// TIA Portal V17 export
// export: Created 2025-11-18T11:18:45.6774883Z, ExportSetting WithDefaults, DisplayName Totally Integrated Automation Portal, DisplayVersion V17 Update 8, DisplayName TIA Portal Openness, DisplayVersion V17 Update 8, DisplayName TIA Portal Version Control Interface, DisplayVersion V17, DisplayName STEP 7 Professional, DisplayVersion V17 Update 8, DisplayName STEP 7 Safety, DisplayVersion V17 Update 6, DisplayName WinCC Advanced, DisplayVersion V17 Update 8
FUNCTION_BLOCK "PLC_VLC_Connection_TCP-IP"   // FB1, LAD
{ S7_Optimized_Access := 'TRUE' }
VERSION : 0.1
// stored: AutoNumber true, IsIECCheckEnabled false, IsRetainMemResEnabled false, MemoryReserve 100, SetENOAutomatically false, UDAEnableTagReadback false
   VAR_INPUT
      xFirstScan : Bool;
      xAlwaysTRUE : Bool;
      xDataReceiveOn : Bool;
   END_VAR
   VAR_OUTPUT
      Connection_OK : Bool;
      Connected : Bool;
      Started : Bool;
      Paused : Bool;
      EndOfFile : Bool;
   END_VAR
   VAR_IN_OUT
      xSendRequest : Bool;
      xCommandStart : Bool;
      xCommandStop : Bool;
      xCommandReset : Bool;
      xCommandPause : Bool;
      xCommandResume : Bool;
      xCommandRewind0 : Bool;
      xCommandRewindX : Bool;
      xReconnect : Bool;
   END_VAR
   VAR
      TCON_Instance { S7_SetPoint := 'True'} : TCON;
      TCON : Struct
         REC : Bool;
         DONE : Bool;
         BUSY : Bool;
         ERROR : Bool;
         DONE_Memo : Bool;
         STATUS : Word;
      END_STRUCT;
      TDISCON : Struct
         REQ : Bool;
         DONE : Bool;
         BUSY : Bool;
         ERROR : Bool;
         STATUS : Word;
      END_STRUCT;
      TSEND : Struct
         REQ : Bool;
         DONE : Bool;
         BUSY : Bool;
         ERROR : Bool;
         DONE_Memo : Bool;
         STATUS : Word;
      END_STRUCT;
      TRCV : Struct
         EN_R : Bool;
         NDR : Bool;
         BUSY : Bool;
         ERROR : Bool;
         STATUS : Word;
         RCVD_LENGTH : UDInt;
      END_STRUCT;
      TDISCON_DB { S7_SetPoint := 'True'} : TDISCON;
      TSEND_Instance { S7_SetPoint := 'True'} : TSEND;
      TRCV_Instance { S7_SetPoint := 'True'} : TRCV;
      Variables : Struct
         ConnectRequest : Bool;
         DisconnectRequest : Bool;
         Reconect : Bool;
         SendString : String;
         DataToSend : String;
         Heartbeat0 : Bool;
         Heartbeat1 : Bool;
         Heartbeat_ConnectionOK : Bool;
         Receive : Array[0..20] of Char;
         ReceivedString : String;
      END_STRUCT;
      Pulses { S7_SetPoint := 'True'} : Array[0..10] of Bool;
      IEC_Timer_SendData { S7_SetPoint := 'True'} : TP_TIME;
      IEC_Timer_SendRequestToLong { S7_SetPoint := 'True'} : TON_TIME;
      IEC_TimerReconnect { S7_SetPoint := 'True'} : TON_TIME;
      IEC_Timer_ReadDelayAfterConnect { S7_SetPoint := 'True'} : TON_TIME;
      TON_HB_1 { S7_SetPoint := 'True'} : TON_TIME;
      TON_HB_2 { S7_SetPoint := 'True'} : TON_TIME;
      TON_HB_3 { S7_SetPoint := 'True'} : TON_TIME;
      ReconnectTimer { S7_SetPoint := 'True'} : TON_TIME;
      RecoonectTimer2 { S7_SetPoint := 'True'} : TON_TIME;
      pulse : Bool;
      pulse2 : Bool;
      resetTimera : Bool;
      pulse3 : Bool;
   END_VAR
   VAR_TEMP
      tempInt : Int;
   END_VAR
   VAR CONSTANT
      EndPoint : String := '\n';
   END_VAR
   VAR_TEMP   // added for the SCL form of the ladder/FBD networks
      _w1 : Bool;
      _w2 : Bool;
      _w3 : Bool;
      _w4 : Bool;
      _w5 : Bool;
      _w6 : Bool;
      _w7 : Bool;
      _w8 : Bool;
      _w9 : Bool;
      _w10 : Bool;
      _w11 : Bool;
      _w12 : Bool;
      _w13 : Bool;
      _w14 : Bool;
      _w15 : Bool;
      _w16 : Bool;
   END_VAR
BEGIN

REGION Network 1: Connection Init
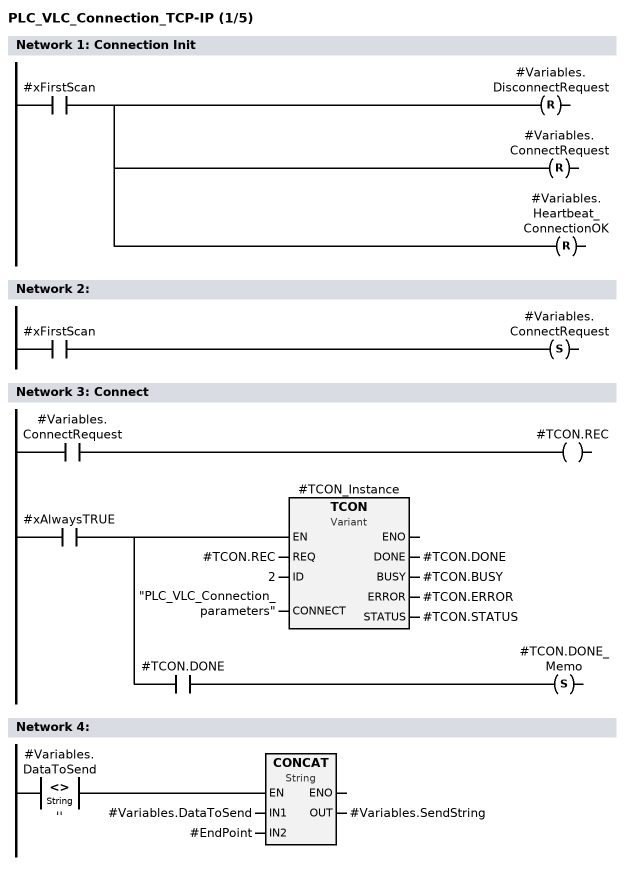
   RUNG wire#powerrail
      Contact( #xFirstScan )
      wire#w1
      R_Coil( #Variables.DisconnectRequest )
   END_RUNG
   RUNG wire#w1
      R_Coil( #Variables.ConnectRequest )
   END_RUNG
   RUNG wire#w1
      R_Coil( #Variables.Heartbeat_ConnectionOK )
   END_RUNG
   // the same network as SCL:
   IF #xFirstScan THEN
       #Variables.DisconnectRequest := FALSE;
       #Variables.ConnectRequest := FALSE;
       #Variables.Heartbeat_ConnectionOK := FALSE;
   END_IF;
END_REGION

REGION Network 2
   RUNG wire#powerrail
      Contact( #xFirstScan )
      S_Coil( #Variables.ConnectRequest )
   END_RUNG
   // the same network as SCL:
   IF #xFirstScan THEN #Variables.ConnectRequest := TRUE; END_IF;
END_REGION

REGION Network 3: Connect
   RUNG wire#powerrail
      Contact( #Variables.ConnectRequest )
      Coil( #TCON.REC )
   END_RUNG
   RUNG wire#powerrail
      Contact( #xAlwaysTRUE )
      wire#w1
      { S7_Templates := "[con_type := Variant, id_type := CONN_OUC]" } #TCON_Instance.TCON(REQ := #TCON.REC, ID := 2, CONNECT := "PLC_VLC_Connection_parameters", DONE => #TCON.DONE, BUSY => #TCON.BUSY, ERROR => #TCON.ERROR, STATUS => #TCON.STATUS)
   END_RUNG
   RUNG wire#w1
      Contact( #TCON.DONE )
      S_Coil( #TCON.DONE_Memo )
   END_RUNG
   // the same network as SCL:
   #TCON.REC := #Variables.ConnectRequest;
   IF #xAlwaysTRUE THEN
       #TCON_Instance(REQ := #TCON.REC,   // TCON
                      ID := 2,
                      CONNECT := "PLC_VLC_Connection_parameters",
                      DONE => #TCON.DONE,
                      BUSY => #TCON.BUSY,
                      ERROR => #TCON.ERROR,
                      STATUS => #TCON.STATUS);
   END_IF;
   IF #xAlwaysTRUE AND #TCON.DONE THEN #TCON.DONE_Memo := TRUE; END_IF;
END_REGION

REGION Network 4
   RUNG wire#powerrail
      { S7_Templates := "SrcType := String" } NE_Contact(in1 := #Variables.DataToSend, in2 := '')
      { S7_Templates := "[card := 2, str_type := String]" } CONCAT(IN1 := #Variables.DataToSend, IN2 := #EndPoint, OUT => #Variables.SendString)
   END_RUNG
   // the same network as SCL:
   IF #Variables.DataToSend <> '' THEN
       CONCAT(IN1 := #Variables.DataToSend, IN2 := #EndPoint, OUT => #Variables.SendString);
   END_IF;
END_REGION

REGION Network 5
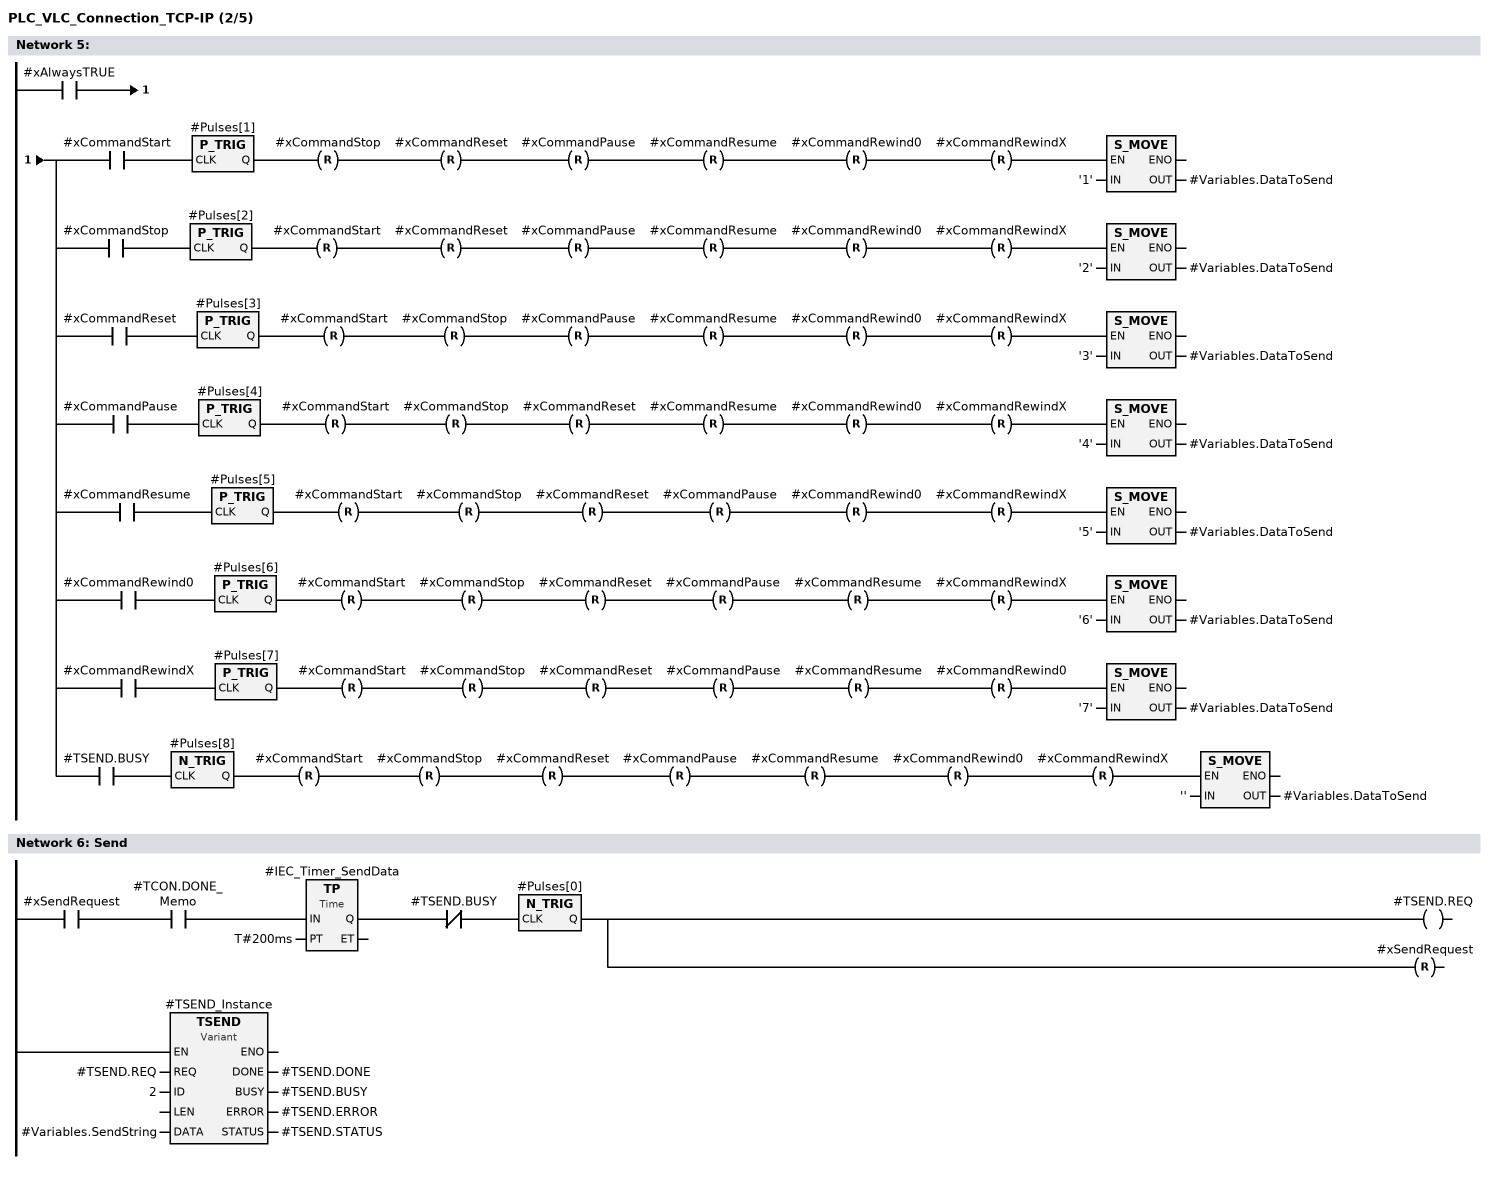
   RUNG wire#powerrail
      Contact( #xAlwaysTRUE )
      wire#w1
      Contact( #xCommandStart )
      P_Trig( #Pulses[1] )
      R_Coil( #xCommandStop )
      R_Coil( #xCommandReset )
      R_Coil( #xCommandPause )
      R_Coil( #xCommandResume )
      R_Coil( #xCommandRewind0 )
      R_Coil( #xCommandRewindX )
      S_Move(in := '1', out => #Variables.DataToSend)
   END_RUNG
   RUNG wire#w1
      Contact( #xCommandStop )
      P_Trig( #Pulses[2] )
      R_Coil( #xCommandStart )
      R_Coil( #xCommandReset )
      R_Coil( #xCommandPause )
      R_Coil( #xCommandResume )
      R_Coil( #xCommandRewind0 )
      R_Coil( #xCommandRewindX )
      S_Move(in := '2', out => #Variables.DataToSend)
   END_RUNG
   RUNG wire#w1
      Contact( #xCommandReset )
      P_Trig( #Pulses[3] )
      R_Coil( #xCommandStart )
      R_Coil( #xCommandStop )
      R_Coil( #xCommandPause )
      R_Coil( #xCommandResume )
      R_Coil( #xCommandRewind0 )
      R_Coil( #xCommandRewindX )
      S_Move(in := '3', out => #Variables.DataToSend)
   END_RUNG
   RUNG wire#w1
      Contact( #xCommandPause )
      P_Trig( #Pulses[4] )
      R_Coil( #xCommandStart )
      R_Coil( #xCommandStop )
      R_Coil( #xCommandReset )
      R_Coil( #xCommandResume )
      R_Coil( #xCommandRewind0 )
      R_Coil( #xCommandRewindX )
      S_Move(in := '4', out => #Variables.DataToSend)
   END_RUNG
   RUNG wire#w1
      Contact( #xCommandResume )
      P_Trig( #Pulses[5] )
      R_Coil( #xCommandStart )
      R_Coil( #xCommandStop )
      R_Coil( #xCommandReset )
      R_Coil( #xCommandPause )
      R_Coil( #xCommandRewind0 )
      R_Coil( #xCommandRewindX )
      S_Move(in := '5', out => #Variables.DataToSend)
   END_RUNG
   RUNG wire#w1
      Contact( #xCommandRewind0 )
      P_Trig( #Pulses[6] )
      R_Coil( #xCommandStart )
      R_Coil( #xCommandStop )
      R_Coil( #xCommandReset )
      R_Coil( #xCommandPause )
      R_Coil( #xCommandResume )
      R_Coil( #xCommandRewindX )
      S_Move(in := '6', out => #Variables.DataToSend)
   END_RUNG
   RUNG wire#w1
      Contact( #xCommandRewindX )
      P_Trig( #Pulses[7] )
      R_Coil( #xCommandStart )
      R_Coil( #xCommandStop )
      R_Coil( #xCommandReset )
      R_Coil( #xCommandPause )
      R_Coil( #xCommandResume )
      R_Coil( #xCommandRewind0 )
      S_Move(in := '7', out => #Variables.DataToSend)
   END_RUNG
   RUNG wire#w1
      Contact( #TSEND.BUSY )
      N_Trig( #Pulses[8] )
      R_Coil( #xCommandStart )
      R_Coil( #xCommandStop )
      R_Coil( #xCommandReset )
      R_Coil( #xCommandPause )
      R_Coil( #xCommandResume )
      R_Coil( #xCommandRewind0 )
      R_Coil( #xCommandRewindX )
      S_Move(in := '', out => #Variables.DataToSend)
   END_RUNG
   // the same network as SCL:
   #_w1 := #xAlwaysTRUE AND #xCommandStart;
   #_w2 := #_w1 AND NOT #Pulses[1];   // rising edge
   #Pulses[1] := #_w1;
   IF #_w2 THEN
       #xCommandStop := FALSE;
       #xCommandReset := FALSE;
       #xCommandPause := FALSE;
       #xCommandResume := FALSE;
       #xCommandRewind0 := FALSE;
       #xCommandRewindX := FALSE;
       #Variables.DataToSend := '1';
   END_IF;
   #_w3 := #xAlwaysTRUE AND #xCommandStop;
   #_w4 := #_w3 AND NOT #Pulses[2];   // rising edge
   #Pulses[2] := #_w3;
   IF #_w4 THEN
       #xCommandStart := FALSE;
       #xCommandReset := FALSE;
       #xCommandPause := FALSE;
       #xCommandResume := FALSE;
       #xCommandRewind0 := FALSE;
       #xCommandRewindX := FALSE;
       #Variables.DataToSend := '2';
   END_IF;
   #_w5 := #xAlwaysTRUE AND #xCommandReset;
   #_w6 := #_w5 AND NOT #Pulses[3];   // rising edge
   #Pulses[3] := #_w5;
   IF #_w6 THEN
       #xCommandStart := FALSE;
       #xCommandStop := FALSE;
       #xCommandPause := FALSE;
       #xCommandResume := FALSE;
       #xCommandRewind0 := FALSE;
       #xCommandRewindX := FALSE;
       #Variables.DataToSend := '3';
   END_IF;
   #_w7 := #xAlwaysTRUE AND #xCommandPause;
   #_w8 := #_w7 AND NOT #Pulses[4];   // rising edge
   #Pulses[4] := #_w7;
   IF #_w8 THEN
       #xCommandStart := FALSE;
       #xCommandStop := FALSE;
       #xCommandReset := FALSE;
       #xCommandResume := FALSE;
       #xCommandRewind0 := FALSE;
       #xCommandRewindX := FALSE;
       #Variables.DataToSend := '4';
   END_IF;
   #_w9 := #xAlwaysTRUE AND #xCommandResume;
   #_w10 := #_w9 AND NOT #Pulses[5];   // rising edge
   #Pulses[5] := #_w9;
   IF #_w10 THEN
       #xCommandStart := FALSE;
       #xCommandStop := FALSE;
       #xCommandReset := FALSE;
       #xCommandPause := FALSE;
       #xCommandRewind0 := FALSE;
       #xCommandRewindX := FALSE;
       #Variables.DataToSend := '5';
   END_IF;
   #_w11 := #xAlwaysTRUE AND #xCommandRewind0;
   #_w12 := #_w11 AND NOT #Pulses[6];   // rising edge
   #Pulses[6] := #_w11;
   IF #_w12 THEN
       #xCommandStart := FALSE;
       #xCommandStop := FALSE;
       #xCommandReset := FALSE;
       #xCommandPause := FALSE;
       #xCommandResume := FALSE;
       #xCommandRewindX := FALSE;
       #Variables.DataToSend := '6';
   END_IF;
   #_w13 := #xAlwaysTRUE AND #xCommandRewindX;
   #_w14 := #_w13 AND NOT #Pulses[7];   // rising edge
   #Pulses[7] := #_w13;
   IF #_w14 THEN
       #xCommandStart := FALSE;
       #xCommandStop := FALSE;
       #xCommandReset := FALSE;
       #xCommandPause := FALSE;
       #xCommandResume := FALSE;
       #xCommandRewind0 := FALSE;
       #Variables.DataToSend := '7';
   END_IF;
   #_w15 := #xAlwaysTRUE AND #TSEND.BUSY;
   #_w16 := NOT #_w15 AND #Pulses[8];   // falling edge
   #Pulses[8] := #_w15;
   IF #_w16 THEN
       #xCommandStart := FALSE;
       #xCommandStop := FALSE;
       #xCommandReset := FALSE;
       #xCommandPause := FALSE;
       #xCommandResume := FALSE;
       #xCommandRewind0 := FALSE;
       #xCommandRewindX := FALSE;
       #Variables.DataToSend := '';
   END_IF;
END_REGION

REGION Network 6: Send
   RUNG wire#powerrail
      Contact( #xSendRequest )
      Contact( #TCON.DONE_Memo )
      { S7_Templates := "time_type := Time" } #IEC_Timer_SendData.TP(pt := T#200ms, et =>)
      I_Contact( #TSEND.BUSY )
      N_Trig( #Pulses[0] )
      wire#w1
      Coil( #TSEND.REQ )
   END_RUNG
   RUNG wire#w1
      R_Coil( #xSendRequest )
   END_RUNG
   RUNG wire#powerrail
      { S7_Templates := "[data_type := Variant, len_type := UDInt, id_type := CONN_OUC]" } #TSEND_Instance.TSEND(REQ := #TSEND.REQ, ID := 2, LEN :=, DATA := #Variables.SendString, DONE => #TSEND.DONE, BUSY => #TSEND.BUSY, ERROR => #TSEND.ERROR, STATUS => #TSEND.STATUS)
   END_RUNG
   // the same network as SCL:
   #IEC_Timer_SendData(IN := #xSendRequest AND #TCON.DONE_Memo, PT := T#200ms);   // TP
   #_w1 := #IEC_Timer_SendData.Q AND NOT #TSEND.BUSY;
   #_w2 := NOT #_w1 AND #Pulses[0];   // falling edge
   #Pulses[0] := #_w1;
   #TSEND.REQ := #_w2;
   IF #_w2 THEN #xSendRequest := FALSE; END_IF;
   #TSEND_Instance(REQ := #TSEND.REQ,   // TSEND
                   ID := 2,
                   DATA := #Variables.SendString,
                   DONE => #TSEND.DONE,
                   BUSY => #TSEND.BUSY,
                   ERROR => #TSEND.ERROR,
                   STATUS => #TSEND.STATUS);
END_REGION

REGION Network 7: Receive
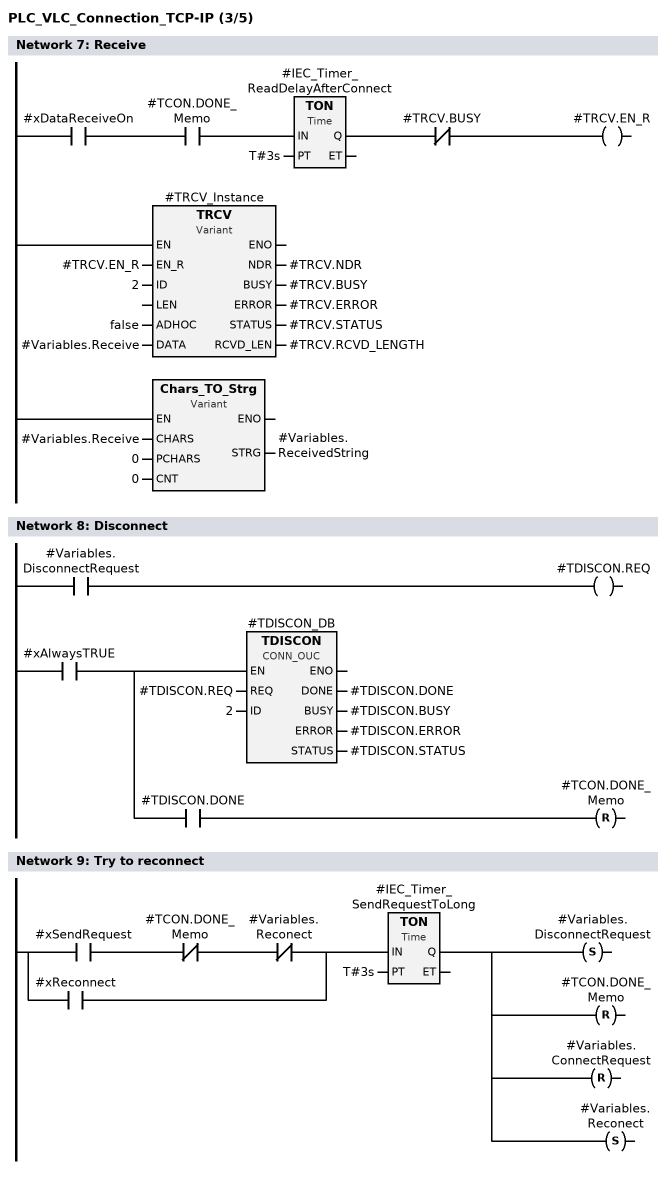
   RUNG wire#powerrail
      Contact( #xDataReceiveOn )
      Contact( #TCON.DONE_Memo )
      { S7_Templates := "time_type := Time" } #IEC_Timer_ReadDelayAfterConnect.TON(pt := T#3s, et =>)
      I_Contact( #TRCV.BUSY )
      Coil( #TRCV.EN_R )
   END_RUNG
   RUNG wire#powerrail
      { S7_Templates := "[card := 1, ptr_type := Variant, value_type := UDInt, id_type := CONN_OUC]" } #TRCV_Instance.TRCV(EN_R := #TRCV.EN_R, ID := 2, LEN :=, ADHOC := false, DATA := #Variables.Receive, NDR => #TRCV.NDR, BUSY => #TRCV.BUSY, ERROR => #TRCV.ERROR, STATUS => #TRCV.STATUS, RCVD_LEN => #TRCV.RCVD_LENGTH)
   END_RUNG
   RUNG wire#powerrail
      { S7_Templates := "[ptr_type := Variant, str_type := String]" } Chars_TO_Strg(Chars := #Variables.Receive, pChars := 0, Cnt := 0, Strg => #Variables.ReceivedString)
   END_RUNG
   // the same network as SCL:
   #IEC_Timer_ReadDelayAfterConnect(IN := #xDataReceiveOn AND #TCON.DONE_Memo, PT := T#3s);   // TON
   #TRCV.EN_R := #IEC_Timer_ReadDelayAfterConnect.Q AND NOT #TRCV.BUSY;
   #TRCV_Instance(EN_R := #TRCV.EN_R,   // TRCV
                  ID := 2,
                  ADHOC := false,
                  DATA := #Variables.Receive,
                  NDR => #TRCV.NDR,
                  BUSY => #TRCV.BUSY,
                  ERROR => #TRCV.ERROR,
                  STATUS => #TRCV.STATUS,
                  RCVD_LEN => #TRCV.RCVD_LENGTH);
   Chars_TO_Strg(Chars := #Variables.Receive, pChars := 0, Cnt := 0, Strg => #Variables.ReceivedString);
END_REGION

REGION Network 8: Disconnect
   RUNG wire#powerrail
      Contact( #Variables.DisconnectRequest )
      Coil( #TDISCON.REQ )
   END_RUNG
   RUNG wire#powerrail
      Contact( #xAlwaysTRUE )
      wire#w1
      { S7_Templates := "id_type := CONN_OUC" } #TDISCON_DB.TDISCON(REQ := #TDISCON.REQ, ID := 2, DONE => #TDISCON.DONE, BUSY => #TDISCON.BUSY, ERROR => #TDISCON.ERROR, STATUS => #TDISCON.STATUS)
   END_RUNG
   RUNG wire#w1
      Contact( #TDISCON.DONE )
      R_Coil( #TCON.DONE_Memo )
   END_RUNG
   // the same network as SCL:
   #TDISCON.REQ := #Variables.DisconnectRequest;
   IF #xAlwaysTRUE THEN
       #TDISCON_DB(REQ := #TDISCON.REQ,   // TDISCON
                   ID := 2,
                   DONE => #TDISCON.DONE,
                   BUSY => #TDISCON.BUSY,
                   ERROR => #TDISCON.ERROR,
                   STATUS => #TDISCON.STATUS);
   END_IF;
   IF #xAlwaysTRUE AND #TDISCON.DONE THEN #TCON.DONE_Memo := FALSE; END_IF;
END_REGION

REGION Network 9: Try to reconnect
   RUNG wire#powerrail
      Contact( #xSendRequest )
      I_Contact( #TCON.DONE_Memo )
      I_Contact( #Variables.Reconect )
      wire#w1
      { S7_Templates := "time_type := Time" } #IEC_Timer_SendRequestToLong.TON(pt := T#3s, et =>)
      wire#w2
      S_Coil( #Variables.DisconnectRequest )
   END_RUNG
   RUNG wire#powerrail
      Contact( #xReconnect )
   END_RUNG wire#w1
   RUNG wire#w2
      R_Coil( #TCON.DONE_Memo )
   END_RUNG
   RUNG wire#w2
      R_Coil( #Variables.ConnectRequest )
   END_RUNG
   RUNG wire#w2
      S_Coil( #Variables.Reconect )
   END_RUNG
   // the same network as SCL:
   #IEC_Timer_SendRequestToLong(IN := (#xSendRequest AND NOT #TCON.DONE_Memo AND NOT #Variables.Reconect) OR #xReconnect,   // TON
                           PT := T#3s);
   IF #IEC_Timer_SendRequestToLong.Q THEN
       #Variables.DisconnectRequest := TRUE;
       #TCON.DONE_Memo := FALSE;
       #Variables.ConnectRequest := FALSE;
       #Variables.Reconect := TRUE;
   END_IF;
END_REGION

REGION Network 10
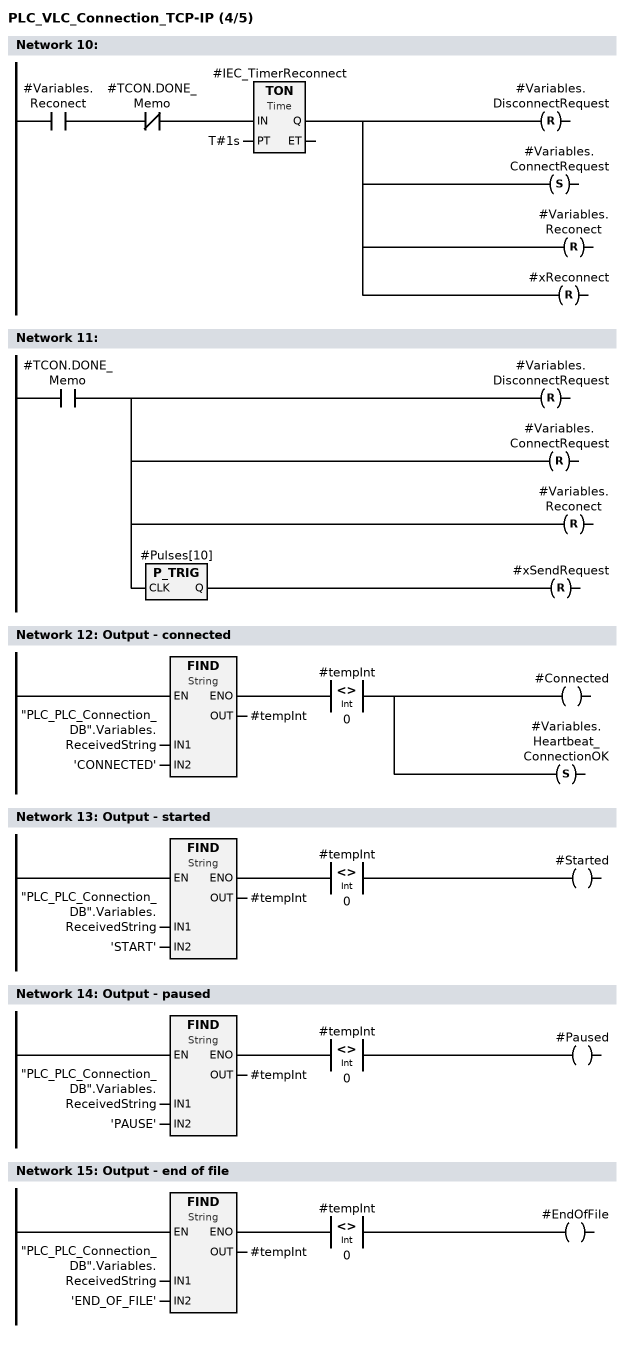
   RUNG wire#powerrail
      Contact( #Variables.Reconect )
      I_Contact( #TCON.DONE_Memo )
      { S7_Templates := "time_type := Time" } #IEC_TimerReconnect.TON(pt := T#1s, et =>)
      wire#w1
      R_Coil( #Variables.DisconnectRequest )
   END_RUNG
   RUNG wire#w1
      S_Coil( #Variables.ConnectRequest )
   END_RUNG
   RUNG wire#w1
      R_Coil( #Variables.Reconect )
   END_RUNG
   RUNG wire#w1
      R_Coil( #xReconnect )
   END_RUNG
   // the same network as SCL:
   #IEC_TimerReconnect(IN := #Variables.Reconect AND NOT #TCON.DONE_Memo, PT := T#1s);   // TON
   IF #IEC_TimerReconnect.Q THEN
       #Variables.DisconnectRequest := FALSE;
       #Variables.ConnectRequest := TRUE;
       #Variables.Reconect := FALSE;
       #xReconnect := FALSE;
   END_IF;
END_REGION

REGION Network 11
   RUNG wire#powerrail
      Contact( #TCON.DONE_Memo )
      wire#w1
      R_Coil( #Variables.DisconnectRequest )
   END_RUNG
   RUNG wire#w1
      R_Coil( #Variables.ConnectRequest )
   END_RUNG
   RUNG wire#w1
      R_Coil( #Variables.Reconect )
   END_RUNG
   RUNG wire#w1
      P_Trig( #Pulses[10] )
      R_Coil( #xSendRequest )
   END_RUNG
   // the same network as SCL:
   IF #TCON.DONE_Memo THEN
       #Variables.DisconnectRequest := FALSE;
       #Variables.ConnectRequest := FALSE;
       #Variables.Reconect := FALSE;
   END_IF;
   #_w1 := #TCON.DONE_Memo AND NOT #Pulses[10];   // rising edge
   #Pulses[10] := #TCON.DONE_Memo;
   IF #_w1 THEN #xSendRequest := FALSE; END_IF;
END_REGION

REGION Network 12: Output - connected
   RUNG wire#powerrail
      { S7_Templates := "str_type := String" } FIND(IN1 := "PLC_PLC_Connection_DB".Variables.ReceivedString, IN2 := 'CONNECTED', OUT => #tempInt)
      { S7_Templates := "SrcType := Int" } NE_Contact(in1 := #tempInt, in2 := 0)
      wire#w1
      Coil( #Connected )
   END_RUNG
   RUNG wire#w1
      S_Coil( #Variables.Heartbeat_ConnectionOK )
   END_RUNG
   // the same network as SCL:
   FIND(IN1 := "PLC_PLC_Connection_DB".Variables.ReceivedString,
        IN2 := 'CONNECTED',
        OUT => #tempInt,
        ENO => #_w1);
   #Connected := #_w1 AND (#tempInt <> 0);
   IF #Connected THEN #Variables.Heartbeat_ConnectionOK := TRUE; END_IF;
END_REGION

REGION Network 13: Output - started
   RUNG wire#powerrail
      { S7_Templates := "str_type := String" } FIND(IN1 := "PLC_PLC_Connection_DB".Variables.ReceivedString, IN2 := 'START', OUT => #tempInt)
      { S7_Templates := "SrcType := Int" } NE_Contact(in1 := #tempInt, in2 := 0)
      Coil( #Started )
   END_RUNG
   // the same network as SCL:
   FIND(IN1 := "PLC_PLC_Connection_DB".Variables.ReceivedString, IN2 := 'START', OUT => #tempInt, ENO => #_w1);
   #Started := #_w1 AND (#tempInt <> 0);
END_REGION

REGION Network 14: Output - paused
   RUNG wire#powerrail
      { S7_Templates := "str_type := String" } FIND(IN1 := "PLC_PLC_Connection_DB".Variables.ReceivedString, IN2 := 'PAUSE', OUT => #tempInt)
      { S7_Templates := "SrcType := Int" } NE_Contact(in1 := #tempInt, in2 := 0)
      Coil( #Paused )
   END_RUNG
   // the same network as SCL:
   FIND(IN1 := "PLC_PLC_Connection_DB".Variables.ReceivedString, IN2 := 'PAUSE', OUT => #tempInt, ENO => #_w1);
   #Paused := #_w1 AND (#tempInt <> 0);
END_REGION

REGION Network 15: Output - end of file
   RUNG wire#powerrail
      { S7_Templates := "str_type := String" } FIND(IN1 := "PLC_PLC_Connection_DB".Variables.ReceivedString, IN2 := 'END_OF_FILE', OUT => #tempInt)
      { S7_Templates := "SrcType := Int" } NE_Contact(in1 := #tempInt, in2 := 0)
      Coil( #EndOfFile )
   END_RUNG
   // the same network as SCL:
   FIND(IN1 := "PLC_PLC_Connection_DB".Variables.ReceivedString,
        IN2 := 'END_OF_FILE',
        OUT => #tempInt,
        ENO => #_w1);
   #EndOfFile := #_w1 AND (#tempInt <> 0);
END_REGION

REGION Network 16: ###########################
END_REGION

REGION Network 17: Communication test - Heartbeat 0
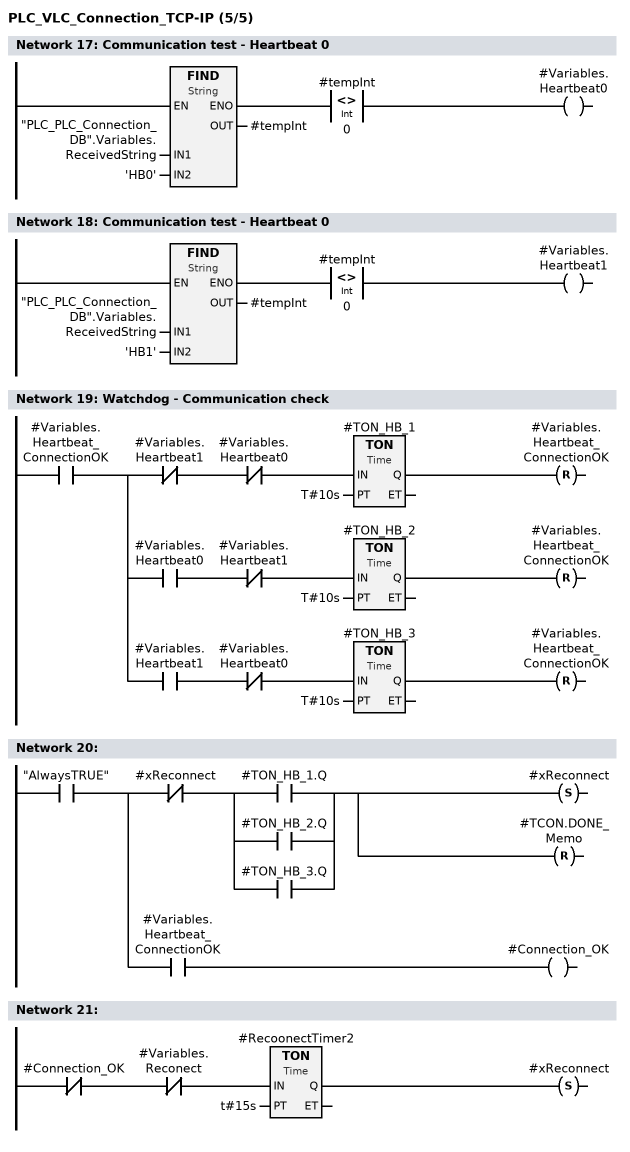
   RUNG wire#powerrail
      { S7_Templates := "str_type := String" } FIND(IN1 := "PLC_PLC_Connection_DB".Variables.ReceivedString, IN2 := 'HB0', OUT => #tempInt)
      { S7_Templates := "SrcType := Int" } NE_Contact(in1 := #tempInt, in2 := 0)
      Coil( #Variables.Heartbeat0 )
   END_RUNG
   // the same network as SCL:
   FIND(IN1 := "PLC_PLC_Connection_DB".Variables.ReceivedString, IN2 := 'HB0', OUT => #tempInt, ENO => #_w1);
   #Variables.Heartbeat0 := #_w1 AND (#tempInt <> 0);
END_REGION

REGION Network 18: Communication test - Heartbeat 0
   RUNG wire#powerrail
      { S7_Templates := "str_type := String" } FIND(IN1 := "PLC_PLC_Connection_DB".Variables.ReceivedString, IN2 := 'HB1', OUT => #tempInt)
      { S7_Templates := "SrcType := Int" } NE_Contact(in1 := #tempInt, in2 := 0)
      Coil( #Variables.Heartbeat1 )
   END_RUNG
   // the same network as SCL:
   FIND(IN1 := "PLC_PLC_Connection_DB".Variables.ReceivedString, IN2 := 'HB1', OUT => #tempInt, ENO => #_w1);
   #Variables.Heartbeat1 := #_w1 AND (#tempInt <> 0);
END_REGION

REGION Network 19: Watchdog - Communication check
   RUNG wire#powerrail
      Contact( #Variables.Heartbeat_ConnectionOK )
      wire#w1
      I_Contact( #Variables.Heartbeat1 )
      I_Contact( #Variables.Heartbeat0 )
      { S7_Templates := "time_type := Time" } #TON_HB_1.TON(pt := T#10s, et =>)
      R_Coil( #Variables.Heartbeat_ConnectionOK )
   END_RUNG
   RUNG wire#w1
      Contact( #Variables.Heartbeat0 )
      I_Contact( #Variables.Heartbeat1 )
      { S7_Templates := "time_type := Time" } #TON_HB_2.TON(pt := T#10s, et =>)
      R_Coil( #Variables.Heartbeat_ConnectionOK )
   END_RUNG
   RUNG wire#w1
      Contact( #Variables.Heartbeat1 )
      I_Contact( #Variables.Heartbeat0 )
      { S7_Templates := "time_type := Time" } #TON_HB_3.TON(pt := T#10s, et =>)
      R_Coil( #Variables.Heartbeat_ConnectionOK )
   END_RUNG
   // the same network as SCL:
   #TON_HB_1(IN := #Variables.Heartbeat_ConnectionOK AND NOT #Variables.Heartbeat1 AND NOT #Variables.Heartbeat0,   // TON
             PT := T#10s);
   #_w1 := #Variables.Heartbeat_ConnectionOK;
   IF #TON_HB_1.Q THEN #Variables.Heartbeat_ConnectionOK := FALSE; END_IF;
   #TON_HB_2(IN := #_w1 AND #Variables.Heartbeat0 AND NOT #Variables.Heartbeat1, PT := T#10s);   // TON
   IF #TON_HB_2.Q THEN #Variables.Heartbeat_ConnectionOK := FALSE; END_IF;
   #TON_HB_3(IN := #_w1 AND #Variables.Heartbeat1 AND NOT #Variables.Heartbeat0, PT := T#10s);   // TON
   IF #TON_HB_3.Q THEN #Variables.Heartbeat_ConnectionOK := FALSE; END_IF;
END_REGION

REGION Network 20
   RUNG wire#powerrail
      Contact( "AlwaysTRUE" )
      wire#w1
      I_Contact( #xReconnect )
      wire#w2
      Contact( #TON_HB_1.Q )
      wire#w3
      S_Coil( #xReconnect )
   END_RUNG
   RUNG wire#w2
      Contact( #TON_HB_2.Q )
   END_RUNG wire#w3
   RUNG wire#w2
      Contact( #TON_HB_3.Q )
   END_RUNG wire#w3
   RUNG wire#w3
      R_Coil( #TCON.DONE_Memo )
   END_RUNG
   RUNG wire#w1
      Contact( #Variables.Heartbeat_ConnectionOK )
      Coil( #Connection_OK )
   END_RUNG
   // the same network as SCL:
   #_w1 := "AlwaysTRUE" AND NOT #xReconnect AND (#TON_HB_1.Q OR #TON_HB_2.Q OR #TON_HB_3.Q);
   IF #_w1 THEN
       #xReconnect := TRUE;
       #TCON.DONE_Memo := FALSE;
   END_IF;
   #Connection_OK := "AlwaysTRUE" AND #Variables.Heartbeat_ConnectionOK;
END_REGION

REGION Network 21
   RUNG wire#powerrail
      I_Contact( #Connection_OK )
      I_Contact( #Variables.Reconect )
      { S7_Templates := "time_type := Time" } #RecoonectTimer2.TON(pt := t#15s, et =>)
      S_Coil( #xReconnect )
   END_RUNG
   // the same network as SCL:
   #RecoonectTimer2(IN := NOT #Connection_OK AND NOT #Variables.Reconect, PT := t#15s);   // TON
   IF #RecoonectTimer2.Q THEN #xReconnect := TRUE; END_IF;
END_REGION
END_FUNCTION_BLOCK
